PROGRAM MAIN
VAR
END_VAR

END_PROGRAM

(* stored: Version 1.1.0.1
   POU MAIN: Id {09667400-14fd-48b0-9895-e96e55090f7a} *)
